FUNCTION_BLOCK FB_PT100 EXTENDS FB_TempSensor IMPLEMENTS I_TempSensor
VAR
	A							: REAL;
	B							: REAL;
	C							: REAL;
END_VAR

(*
	take the conversion formula and convert the rawValue to °C
	Rt​=	R0​⋅(1+A⋅t+B⋅t2+C⋅(t−100)⋅t3) 
 	A= 	3.9083⋅10−3
	B= 	−5.7750⋅10−7
	C=	−4.1830⋅10	for t​<​0°C
		−120.0		for t​≥​0°C
*)
_degrees := rawValue + 100.0;

END_FUNCTION_BLOCK

(* stored: Version 1.1.0.1, ProductVersion 3.1.4024.12
   POU FB_PT100: Id {4cddf425-4391-4091-a74f-15d20369c1a0}, SpecialFunc None *)
